// TIA Portal V19 export
TYPE "LAF_typeHeaderPlcToHmi"
// Information from the PLC to the HMI
// stored: Access Published
   STRUCT
      powerStatus { ExternalWritable := 'False'} : Int;   // 0 - Off, 1 - Paused, 2 - On
      displayedMode { ExternalWritable := 'False'} : DInt;   // Current mode according to the units selected
      displayedState { ExternalWritable := 'False'} : DInt;   // Current state according to the units selected
      modeRequestsButtons { ExternalWritable := 'False'} : "LUC_typeButtons";   // Set properties of the mode request buttons
      stateCommandsButtons { ExternalWritable := 'False'} : "LUC_typeButtons";   // Set properties of the state commands buttons
      specialFunctionButtons { ExternalWritable := 'False'} : "LUC_typeButtons";   // Set properties of the special functions buttons
   END_STRUCT;
END_TYPE
